// TwinCAT 3 PLC project NCAxisDemo
// ProgramVersion: 3.1.4023.0
// libraries:
//   Tc2_MC2, * (Beckhoff Automation GmbH)
//   Tc2_Standard, * (Beckhoff Automation GmbH)
//   Tc2_System, * (Beckhoff Automation GmbH)
//   Tc3_Module, * (Beckhoff Automation GmbH)
// project tree:
//   / PlcTask.TcTTO
//   POUs/AxisManager/ FB_Axis.TcPOU
//   POUs/Blinker/ FB_Blinker.TcPOU
//   POUs/ MAIN.TcPOU
// real-time tasks:
//   TASK PlcTask: cycle T#10ms, priority 20, ADS port 350
// motion (NC):
//   TASK NC-Task 1 SAF: cycle T#2ms, priority 4, ADS port 501
//   TASK NC-Task 1 SVB: cycle T#10ms, priority 8, ADS port 511
//   AXIS Axis 1 (id 1)
//     OtherSettings: AllowMotionCmdToSlave=true
//     encoder EncType=1
//     drive DrvType=5
//       Analog: TorqueSetpointScale=10, ScaleFactorActTorque=0.1
//     controller CtrType=1
//       CtrPara: PriorControlFactor=1
//         Observer: BandWidth=20
// variable links:
//   NCAxisDemo Instance <-> NC-Task 1 SAF/Axes/Axis 1
//     PlcTask Inputs/MAIN.stAxisRef.NcToPlc <-> Outputs/ToPlc
//     PlcTask Outputs/MAIN.stAxisRef.PlcToNc <-> Inputs/FromPlc

CONFIGURATION NCAxisDemo
    RESOURCE PLC ON TwinCAT3
        TASK PlcTask(INTERVAL := T#10ms, PRIORITY := 20);
        PROGRAM MAIN WITH PlcTask : MAIN;
    END_RESOURCE
END_CONFIGURATION

// ---- POUs/MAIN.TcPOU
PROGRAM MAIN
VAR

	stAxisRef	: AXIS_REF;		// Axis reference for our demo motion axis
	fbAxis		: FB_Axis;		// Instance of our axis management FB

	// Axis state outputs
	bAxisReady	: BOOL;			// Set when the axis is enable and ready for motion 
	bError		: BOOL;			// Set when the axis or the internal MC functions have an error

	
	// Bools to activate different tests
	bTestEnable	: BOOL;			// Set to enable the axis 
	bTestDisable: BOOL;			// Set to disable the axis 
	bTestReset	: BOOL;			// Set to reset the axis 
	bTestRecal	: BOOL;			// Set to reset the axis position
	bTestStop	: BOOL;			// Set to perform a blocking stop on the axis 
	bTestDynamicVelocity: BOOL;	// Test sending a dynamically updating target speed to the axis 
	
	
	fbBlinker	: FB_Blinker;	// Used to generate a changing velocity signal for the test

END_VAR

// We run the axis managment FB every cycle
fbAxis(	AxisRef		:= stAxisRef,
		bAxisReady	=>bAxisReady,
		bError		=> bError);

// Also run the blinker to generate a target velocity signal	
fbBlinker(Period	:= T#2S);

// Run different tests of the Axis Management FB functionality.
	
IF(bTestEnable)THEN
	bTestEnable:=FALSE;
	fbAxis.Enable();
END_IF

IF(bTestDisable)THEN
	bTestDisable:=FALSE;
	fbAxis.Disable();
END_IF

IF(bTestReset)THEN
	bTestReset:=FALSE;
	fbAxis.Reset();
END_IF

IF(bTestRecal)THEN
	bTestRecal:=FALSE;
	fbAxis.ResetPosition(fPosition:=100);
END_IF

IF(bTestStop)THEN
	bTestStop:=FALSE;
	fbAxis.Stop();
END_IF

// Test Dynamic velocity
IF(bTestDynamicVelocity) THEN
	fbAxis.DynamicVelocity(fVelocity:=fbBlinker.fET);
END_IF

END_PROGRAM

// ---- POUs/AxisManager/FB_Axis.TcPOU
FUNCTION_BLOCK FB_Axis
VAR_INPUT
END_VAR
VAR_IN_OUT
	AxisRef	: AXIS_REF;
END_VAR
VAR_OUTPUT
	bDynamicVelocityActive	: BOOL;
	bAxisReady				: BOOL;
	bError					: BOOL;
END_VAR
VAR
	//AxisRef		: AXIS_REF;

	bReset			: BOOL;			// Rising edge triggers  reset 
	bReCalibrate	: BOOL;			// Rising edge triggers axis position reset 
	fCalPosition	: LREAL;		// The calibration position
	bPowerOn		: BOOL;			// Enable, keep high for axis enable
	bNotFastDisable	: BOOL	:= TRUE;// Used for the hard fault disable
	bDelayPowerOff	: BOOL;			// Used for controlled axis stop.
	bStopAxis		: BOOL;			// Used for controlled axis stop

	
	fbReadAxisParam		: MC_ReadParameter;	// FB to get axis max Decel
	fAxisMaxDec			: LREAL;	// The max axis Deceleration, read from the axis config

	// Motion axis functions
	McPower	: MC_Power;
	McReset	: MC_Reset;
	McHome	: MC_Home;
	
	// Edge detection 
	fbReCalibrate			: TP;
	fbExtReset				: TP;
	fbGetAxisParam			: TP;
	fbFallingExtResetQ		: F_TRIG;
	fbFallingRecalibrateQ	: F_TRIG;
	fbFallingPowerOn		: F_TRIG;
	fbRisingMcPowerStatus	: R_TRIG;
	fbRisingMcResetDone		: R_TRIG;
	fbRisingMcHomeDone		: R_TRIG;
	fbRisingStopDone		: R_TRIG;
	fbRisingHaltDone		: R_TRIG;
	fbRisingPowerON			: R_TRIG;
	
	// Distinguish between standard home and special home
	iHomeSource	: INT	:= 1; // 1 for startup home, 2 for other home function 
	
	// Dynamic velocity
	fDynamicVelo			: LREAL;
	fbFallingDynamicVelocity: F_TRIG;
	bPhase					: BOOL;
	bDvHeartBeat			: BOOL;
	bDelayHaltDisable		: BOOL;
	bBlockDynamicVelocity	: BOOL;
	McMoveVelocity_A		: MC_MoveVelocity;
	McMoveVelocity_B		: MC_MoveVelocity;
	McHalt					: MC_Halt;
	McStop					: MC_Stop;
	
	eMotionDirection		: MC_Direction;
	
	
END_VAR

// Run edge detection FB's (AXIS MANAGENEMT) 
fbRisingMcPowerStatus(CLK:=McPower.Status);
fbRisingPowerON(CLK:=bPowerOn);
fbRisingMcResetDone(CLK:=McReset.Done);
fbRisingMcHomeDone(CLK:=McHome.Done);
fbExtReset(IN:=bReset,PT:=T#2MS);
fbFallingExtResetQ(CLK:=fbExtReset.Q);
fbReCalibrate(IN:=bReCalibrate,PT:=T#2MS);
fbFallingRecalibrateQ(CLK:=fbReCalibrate.Q);
fbFallingPowerOn(CLK:=bPowerOn);
fbGetAxisParam(IN:=fbRisingMcPowerStatus.Q,PT:=T#20MS);
fbRisingStopDone(CLK:=McStop.Done);
fbRisingHaltDone(CLK:=McHalt.Done);

// Run edge detection FB's (DYNAMIC VELOCITY) 
fbFallingDynamicVelocity(CLK:=bDynamicVelocityActive);

// Delay the HALT disable to allow axis to halt when disabling dynamic velocity mode
IF(fbFallingDynamicVelocity.Q)THEN
	bDelayHaltDisable	:= TRUE;
END_IF

IF(fbRisingMcResetDone.Q) THEN
	bBlockDynamicVelocity	:= FALSE;
END_IF


IF(fbRisingStopDone.Q)THEN
	bStopAxis		:= FALSE;
	bDelayPowerOff	:= FALSE;
END_IF

IF(fbFallingPowerOn.Q)THEN
	IF(AxisRef.NcToPlc.AxisState <> 0)THEN
		bStopAxis		:= TRUE;			// trigger a controlled axis stop if the axis is disabled while running a motion
		bDelayPowerOff	:= TRUE;			// Delay the power off until the axis has come to a stop
	END_IF
END_IF

IF(fbFallingExtResetQ.Q)THEN
	bReset	:= FALSE;
END_IF

IF(fbFallingRecalibrateQ.Q)THEN
	bReCalibrate	:= FALSE;
END_IF

// Read the Max Deceleration from the axis 
fbReadAxisParam(	Axis			:= AxisRef, 
					Enable			:= fbGetAxisParam.Q,
					ParameterNumber	:= MC_AxisParameter.AxisMaximumDeceleration,
					Value			=> fAxisMaxDec);

//Check for errors 
IF(	(McPower.Error) OR 
	(McReset.Error) OR 
	(McHome.Error)	OR
	(AxisRef.NcToPlc.ErrorCode <> 0)) THEN
	
		bError := TRUE;
	
	ELSE
		bError := FALSE;
END_IF

// Run MC Power, Reset and Home Functions
McPower(	Axis			:= AxisRef,
			Enable			:= (bDelayPowerOff OR bPowerOn) AND bNotFastDisable,
			Enable_Positive	:= TRUE,
			Enable_Negative	:= TRUE,
			Override		:= 100);
			
McReset( 	Axis			:= AxisRef,
			Execute			:= (fbRisingMcPowerStatus.Q OR fbExtReset.Q OR (fbRisingPowerON.Q AND (AxisRef.NcToPlc.ErrorCode <> 0)) ));
// Home
CASE iHomeSource OF 
	1:	
		// standard start up force calibration 
		McHome( 	Axis			:= AxisRef,
					HomingMode		:= MC_HomingMode.MC_ForceCalibration,
					Execute			:= fbRisingMcResetDone.Q);
	2: 
		// recalibration function direct calibration 
		McHome( 	Axis			:= AxisRef,
					HomingMode		:= MC_HomingMode.MC_Direct,
					Position		:= fCalPosition,
					Execute			:= fbReCalibrate.Q);
	ELSE
		iHomeSource	:= 1;
END_CASE	


// Swap back to default home source when home completes
IF(fbRisingMcHomeDone.Q)THEN
	iHomeSource	:= 1;
END_IF	

// Set the output axis ready flag					
IF(bPowerOn AND fbRisingMcHomeDone.Q AND NOT(bError))THEN
	bAxisReady	:= TRUE;
END_IF		

// Reset the output axis ready flag 
IF(NOT(bPowerOn) OR bError)THEN
	bAxisReady	:= FALSE;	
END_IF



// Dynamic Velocity Implementation
IF(bDynamicVelocityActive AND NOT(bBlockDynamicVelocity)) THEN
	
	bPhase	:= NOT(bPhase);	// Phase alternator to allow continuous target velocity updates
	
	McMoveVelocity_A( 	Axis			:= AxisRef,
						Execute			:= (bPhase AND (fDynamicVelo <> 0) AND bPowerOn),
						Direction		:= eMotionDirection,
						Velocity		:= ABS(fDynamicVelo));
	
	McMoveVelocity_B( 	Axis			:= AxisRef,
						Execute			:= (NOT(bPhase) AND (fDynamicVelo <> 0) AND bPowerOn),
						Direction		:= eMotionDirection,
						Velocity		:= ABS(fDynamicVelo));
	
	
	// Run a heartbeat to disablle dynamic velocity as soon as the user stops updating it					
	IF(NOT(bDvHeartBeat))THEN
		bDynamicVelocityActive	:= FALSE;
	END_IF
	
	// Reset the dynamic velocity active state
	bDvHeartBeat	:= FALSE;
	
						
END_IF 

IF(bDynamicVelocityActive OR bDelayHaltDisable) THEN
	// This is used for dynamic velocity mode 
	McHalt			(	Axis			:= AxisRef,
						Deceleration	:= fAxisMaxDec,
						Execute			:= ((fDynamicVelo = 0) AND bPowerOn) OR fbFallingDynamicVelocity.Q);
	
	// reset bDelay halt disable when the halt function completes 
	IF(fbRisingHaltDone.Q)THEN
		bDelayHaltDisable	:= FALSE;
	END_IF
						
END_IF

// Implement a max dec controller axis Stop if the axis is disabled while running a motion
McStop			(	Axis			:= AxisRef,
					Deceleration	:= fAxisMaxDec,
					Execute			:= bStopAxis);

METHOD Disable : BOOL // Disbales the axis after stopping the axis as fast as possible , graceful stop 
VAR_INPUT
END_VAR
THIS^.bPowerOn				:= FALSE;
END_METHOD

METHOD DynamicVelocity : BOOL
VAR_INPUT
	fVelocity	: LREAL;
END_VAR
IF(THIS^.bAxisReady) THEN 
	IF(NOT(bDynamicVelocityActive)) THEN THIS^.bDynamicVelocityActive := TRUE; END_IF // Assert the dynamic velocity active flag 
	THIS^.bDvHeartBeat 			:= TRUE;		// Run the dynamic velocity active heartbeat 
	THIS^.fDynamicVelo			:= fVelocity;	// Update the target velocity
	IF(fVelocity > 0)THEN
		THIS^.eMotionDirection	:= MC_Direction.MC_Positive_Direction;
	ELSE
		THIS^.eMotionDirection	:= MC_Direction.MC_Negative_Direction;
	END_IF
END_IF
END_METHOD

METHOD Enable : BOOL
VAR_INPUT
END_VAR
THIS^.bPowerOn					:= TRUE;
THIS^.bNotFastDisable			:= TRUE;
THIS^.bDynamicVelocityActive	:= FALSE;
END_METHOD

METHOD FastDisable : BOOL	// Disbales the axis immediately, if moving will result in a fault
VAR_INPUT
END_VAR
THIS^.bNotFastDisable	:= FALSE;
END_METHOD

METHOD Reset : BOOL
VAR_INPUT
END_VAR
THIS^.bReset					:= TRUE;
THIS^.bDynamicVelocityActive	:= FALSE;
END_METHOD

METHOD ResetPosition : BOOL
VAR_INPUT
	fPosition	: LREAL; 	// Calibration axis position 
END_VAR
bReCalibrate		:= TRUE;
fCalPosition		:= fPosition;
THIS^.iHomeSource	:= 2;
END_METHOD

METHOD Stop : BOOL
VAR_INPUT
END_VAR
THIS^.bStopAxis					:= TRUE;
THIS^.bBlockDynamicVelocity		:= TRUE;
END_METHOD

END_FUNCTION_BLOCK

// ---- POUs/Blinker/FB_Blinker.TcPOU
FUNCTION_BLOCK FB_Blinker
VAR_INPUT
	Period	: TIME;
END_VAR
VAR_OUTPUT
	Output	: BOOL;
	fET		: LREAL;
END_VAR
VAR
	Timer1: TON;
END_VAR

Timer1(In := NOT Timer1.Q, PT := Period);
Output	:= Period/2 > Timer1.ET;
fET		:= TIME_TO_LREAL(Timer1.ET);

END_FUNCTION_BLOCK
